// TIA Portal V20 export
// export: Created 2026-04-11T06:02:29.7812473Z, ExportSetting WithDefaults, DisplayName Totally Integrated Automation Portal, DisplayVersion V20, DisplayName TIA Portal Openness, DisplayVersion V20, DisplayName TIA Portal Version Control Interface, DisplayVersion V20, DisplayName STEP 7 Professional, DisplayVersion V20, DisplayName STEP 7 Safety, DisplayVersion V20, DisplayName WinCC Basic/Comfort/Advanced, DisplayVersion V20, DisplayName WinCC Unified, DisplayVersion V20
TYPE "udtContC_S"
// stored: IsFailsafeCompliant false
   STRUCT
      LMN : Real;
      LMN_PER : Word;
      QLMN_HLM : Bool;
      QLMN_LLM : Bool;
      LMN_P : Real;
      LMN_I : Real;
      LMN_D : Real;
      PV : Real;
      ER : Real;
   END_STRUCT;
END_TYPE
